// TIA Portal V20 export
// export: Created 2025-12-01T14:57:11.2126778Z, ExportSetting None, DisplayName Totally Integrated Automation Portal, DisplayVersion V20 Update 3, DisplayName TIA Portal Openness, DisplayVersion V20 Update 3, DisplayName TIA Portal Version Control Interface, DisplayVersion V20 Update 3, DisplayName STEP 7 Professional, DisplayVersion V20 Update 3, DisplayName STEP 7 Safety, DisplayVersion V20 Update 2, DisplayName WinCC Basic/Comfort/Advanced, DisplayVersion V20 Update 3, DisplayName WinCC Professional, DisplayVersion V20 Update 3, DisplayName WinCC Unified, DisplayVersion V20 Update 3
FUNCTION "FC505_CNT_ET_OK_NOOK" : Void   // FC505, LAD
{ S7_Optimized_Access := 'FALSE' }
AUTHOR : TLigero
NAME : 20130623
VERSION : 3.1
// stored: AutoNumber false, SetENOAutomatically false
   VAR_INPUT
      Num_Scanner : UInt;
      Evento_a_Registrar : UInt;   // 1 lectura nook, 2 lectura ok, 3 lectura no encontrada
   END_VAR
   VAR_TEMP
      Cero : Byte;
      retval : Int;
      Auxiliar : UInt;
   END_VAR
BEGIN

NETWORK
TITLE = inicializacion
//============================================================

      L     0;
      T     #Cero;


//============================================================

NETWORK
TITLE = Sacamos los datos previamente guardados para actualizarlos
//============================================================
// -- revisamos si hay algún dato que se va a desbordar

      SET;
      L     "DB216_Cnt_Estadisticas_Scanners".CNT_LectSCR[#Num_Scanner].Lect_Good;
      L     65535;
      ==I;
      JC    inicializa;


      SET;
      L     "DB216_Cnt_Estadisticas_Scanners".CNT_LectSCR[#Num_Scanner].Lect_NoGood;
      L     65535;
      ==I;
      JC    inicializa;

      JU    registra_datos;

//============================================================
// -- Ponemos a cero todos los datos salvo el contador
// -- de lecturas malas consecutivas
inicializa:NOP   0;

      L     "DB216_Cnt_Estadisticas_Scanners".CNT_LectSCR[#Num_Scanner].Lect_NoGood_consecutivas;
      T     #Auxiliar;
      CALL  FILL
      ( BVAL    := #Cero,
        RET_VAL := #retval,
        BLK     := "DB216_Cnt_Estadisticas_Scanners".CNT_LectSCR[#Num_Scanner]
      );

      L     #Auxiliar;
      T     "DB216_Cnt_Estadisticas_Scanners".CNT_LectSCR[#Num_Scanner].Lect_NoGood_consecutivas;
//============================================================


NETWORK
TITLE = Registrar los datos
//============================================================
registra_datos:NOP   0;

      L     #Evento_a_Registrar;

      JL    valor_no_valido;

      JU    valor_no_valido;  // --- Con dato 0
      JU    contar_lectura_nook;  // --- Con dato 1
      JU    contar_lectura_ok;  // --- Con dato 2
      JU    contar_no_encontradas;  // --- Con dato 2

valor_no_valido:JU    guardar_datos;  // --- Motivo INEXISTENTE


//============================================================
// -- Contar lectura ok

contar_lectura_nook:NOP   0;
      L     "DB216_Cnt_Estadisticas_Scanners".CNT_LectSCR[#Num_Scanner].Lect_NoGood;
      L     1;
      +I;
      T     "DB216_Cnt_Estadisticas_Scanners".CNT_LectSCR[#Num_Scanner].Lect_NoGood;

//-- incrementamos también el contador
// -- de lecturas malas consecutivas
      L     "DB216_Cnt_Estadisticas_Scanners".CNT_LectSCR[#Num_Scanner].Lect_NoGood_consecutivas;
      L     1;
      +I;
      T     "DB216_Cnt_Estadisticas_Scanners".CNT_LectSCR[#Num_Scanner].Lect_NoGood_consecutivas;

      JU    guardar_datos;

//============================================================
// -- Contar lectura ok

contar_lectura_ok:NOP   0;
      L     "DB216_Cnt_Estadisticas_Scanners".CNT_LectSCR[#Num_Scanner].Lect_Good;
      L     1;
      +I;
      T     "DB216_Cnt_Estadisticas_Scanners".CNT_LectSCR[#Num_Scanner].Lect_Good;

//-- como hemos tenido lectura ok
//-- reseteamos el contador de errores consecutivos
      L     0;
      T     "DB216_Cnt_Estadisticas_Scanners".CNT_LectSCR[#Num_Scanner].Lect_NoGood_consecutivas;

      JU    guardar_datos;
//============================================================
// -- Contar no encontrada
// -- Suma 1 también a lectura ok
contar_no_encontradas:NOP   0;

      L     "DB216_Cnt_Estadisticas_Scanners".CNT_LectSCR[#Num_Scanner].Lect_NoFound;
      L     1;
      +I;
      T     "DB216_Cnt_Estadisticas_Scanners".CNT_LectSCR[#Num_Scanner].Lect_NoFound;

      L     "DB216_Cnt_Estadisticas_Scanners".CNT_LectSCR[#Num_Scanner].Lect_Good;
      L     1;
      +I;
      T     "DB216_Cnt_Estadisticas_Scanners".CNT_LectSCR[#Num_Scanner].Lect_Good;

//-- como hemos tenido lectura ok
//-- reseteamos el contador de errores consecutivos
      L     0;
      T     "DB216_Cnt_Estadisticas_Scanners".CNT_LectSCR[#Num_Scanner].Lect_NoGood_consecutivas;

      JU    guardar_datos;

//============================================================

NETWORK
TITLE = Guardar los datos actualizados
//============================================================
guardar_datos:NOP   0;


//============================================================

END_FUNCTION
